// TIA Portal V20 export
DATA_BLOCK "ToteDir"   // DB43
// stored: MemoryReserve 100, Namespace EmptyLine
   VAR
      Conveyor : Array[_."J1.6.1".._."J1.6.2"] of "Global.ItemDir";
   END_VAR
BEGIN
END_DATA_BLOCK
